TYPE SAI_Feedback :
STRUCT
	{attribute addProperty Name "Settings"}
	Settings AT %I* : SAI_Feedback_Settings;
END_STRUCT
END_TYPE

(* stored: Version 1.1.0.1, ProductVersion 3.1.4024.9
   DUT SAI_Feedback: Id {4d125d2a-3cf7-07a8-0d88-ae0644a0bad8} *)
